FUNCTION INTERNAL F_LogError : BOOL
VAR_INPUT
    Source  : T_MaxString;
    Message : T_MaxString;
END_VAR
VAR
END_VAR

ADSLOGSTR(msgCtrlMask := ADSLOG_MSGTYPE_STRING OR ADSLOG_MSGTYPE_ERROR OR ADSLOG_MSGTYPE_LOG OR ADSLOG_MSGTYPE_MSGBOX,
          msgFmtStr   := FormatStringEx2('%s : %s', Source, Message),
          strArg      := '');

END_FUNCTION

(* stored: Version 1.1.0.1, ProductVersion 3.1.4024.12
   POU F_LogError: Id {737d3fea-66b0-40d3-b566-1b8aff3a3a7f}, SpecialFunc None *)
